{attribute 'qualified_only'}
VAR_GLOBAL
END_VAR

(* stored: Version 1.1.0.1, ProductVersion 3.1.4024.6
   GVL synGlobal: Id {11dc25b2-c732-4417-9e7f-47504976b06f} *)
